TYPE ST_Euchner_MSM_HW_IN :
STRUCT
	///Hardware In
	nByte0: USINT;
END_STRUCT
END_TYPE

(* stored: Version 1.1.0.1, ProductVersion 3.1.4024.12
   DUT ST_Euchner_MSM_HW_IN: Id {7ac167dc-ca70-44a4-b886-d4046fec814b} *)
